// TwinCAT 3 PLC project IOLink
// Title: TcUnit advanced example
// Company: www.tcunit.org
// Author: Jakob Sagatowski
// ProjectVersion: 1.0.0.0
// Description: This library is a demonstration of the TcUnit framework, which is a TwinCAT unit testing framework. It implements certain parts of the IO-Link functionality. IO-Link is a serial communication protocol for end devices such as various types of sensors (temperature, pressure, etc) and actuators. The functionality implemented in this library is related to the "diagnosis" part of IO-Link, which in EtherCAT masters is implemented using the diagnosis history object defined in the ETG1020 specification.
// ProgramVersion: 3.1.4022.7
// libraries:
//   Tc2_EtherCAT, * (Beckhoff Automation GmbH)
//   Tc2_Standard, * (Beckhoff Automation GmbH)
//   Tc2_System, * (Beckhoff Automation GmbH)
//   Tc3_Module, * (Beckhoff Automation GmbH)
//   TcUnit, * (www.tcunit.org)
// project tree:
//   DUTs/ E_DIAGNOSISTYPE.TcDUT (not stored), E_DIAGNOSTICCODETYPE.TcDUT (not stored), E_EVENTQUALIFIERMODE.TcDUT (not stored), E_TIMESTAMPTYPE.TcDUT (not stored), ST_DIAGNOSTICCODE.TcDUT (not stored), ST_DIAGNOSTICMESSAGE.TcDUT (not stored), ST_FLAGS.TcDUT (not stored)
//   / PlcTask.TcTTO (not stored)
//   POUs/ FB_DiagnosticMessageDiagnosticCodeParser.TcPOU (not stored), FB_DiagnosticMessageFlagsParser.TcPOU (not stored), FB_DiagnosticMessageParser.TcPOU (not stored), FB_DiagnosticMessageTextIdentityParser.TcPOU (not stored), FB_DiagnosticMessageTimeStampParser.TcPOU (not stored), F_DWORDFromBytes.TcPOU (not stored), F_WORDFromBytes.TcPOU (not stored)
//   Test/ FB_DiagnosticMessageDiagnosticCodeParser_Test.TcPOU (not stored), FB_DiagnosticMessageFlagsParser_Test.TcPOU (not stored), FB_DiagnosticMessageParser_Test.TcPOU (not stored), FB_DiagnosticMessageTextIdentityParser_Test.TcPOU (not stored), FB_DiagnosticMessageTimeStampParser_Test.TcPOU (not stored), PRG_TEST.TcPOU
// real-time tasks:
//   TASK PlcTask: cycle T#10ms, priority 20, ADS port 350

// ---- Test/PRG_TEST.TcPOU
(*
    This is the main program for execution of the unit tests.
	This is the main program for execution of the unit tests.
	This is the main program for execution of the unit tests.
	This is the main program for execution of the unit tests.
	This is the main program for execution of the unit tests.
*)
PROGRAM PRG_TEST
VAR	
    (* Test function blocks *)
    fbDiagnosticMessageDiagnosticCodeParser_Test : FB_DiagnosticMessageDiagnosticCodeParser_Test;
    fbDiagnosticMessageFlagsParser_Test : FB_DiagnosticMessageFlagsParser_Test;
    fbDiagnosticMessageParser_Test : FB_DiagnosticMessageParser_Test;
    fbDiagnosticMessageTextIdentityParser_Test : FB_DiagnosticMessageTextIdentityParser_Test;
    fbDiagnosticMessageTimeStampParser_Test : FB_DiagnosticMessageTimeStampParser_Test;
END_VAR

TcUnit.RUN();

END_PROGRAM
